FUNCTION TFDirezioneAssePositiva : BOOL (*Valuta la direzione dell'asse in base alla sua quota attuale e alla sua destinazione*)
VAR_INPUT
	Posizione_Attuale 	: LREAL; //Posizione in cui si trova l'Asse
	Posizione_Finale 	: LREAL; //Posizione finale di posizionamento dell'Asse
END_VAR
VAR
END_VAR
(*Valuta la direzione dell'asse in base alla sua quota attuale e alla sua destinazione*)

TFDirezioneAssePositiva := FALSE;
IF Posizione_Attuale < Posizione_Finale THEN
	TFDirezioneAssePositiva := TRUE;
	RETURN;
END_IF

END_FUNCTION

(* stored: Version 1.1.0.1, ProductVersion 3.1.4024.11
   POU TFDirezioneAssePositiva: Id {84bed7a7-8de3-4255-9b76-8479445a2cd7}, SpecialFunc None *)
